GLOBALCONSTANTS AID_DM (* Data mask object attribute ids *)
  (* Standard: 61499-1; Description: Copyright (c) 2023 HR Agrartechnik GmbH This program and the accompanying materials are made available under the terms of the Eclipse Public License 2.0 which is available at https://www.eclipse.org/legal/epl-2.0/ SPDX-License-Identifier: EPL-2.0 *)
  (* Version 1.0, 2026-06-20, Franz Höpfinger, HR Agrartechnik GmbH *)
  PACKAGE isobus::UT::Q::const::AID;
  IMPORT eclipse4diac::core::TypeHash;
  VAR_GLOBAL CONSTANT
    BACKGROUND_COLOUR : USINT := USINT#1; (* 1: AID_DM_BACKGROUND_COLOUR - Background colour index. *)
    SOFT_KEY_MASK : USINT := USINT#2; (* 2: AID_DM_SOFT_KEY_MASK - Object ID of a Soft Key Mask associated with this Data Mask. *)
  END_VAR
END_GLOBALCONSTANTS
